{attribute 'GeneratedUsingTerminal: EK1100-0000-0018'}
{attribute addProperty BoxType "EK1100-0000-0018"}
{attribute addProperty Id "RC20_B1_EL7041_1000EL7041_86DE63E743RC20_B2_EL7041_1000EL7041_86DE63E743RC20_C11_EL7041_1000EL7041_86DE63E743RC20_C12_EL7041_1000EL7041_86DE63E743RC20_C21_EL7041_1000EL7041_86DE63E743RC20_C22_EL7041_1000EL7041_86DE63E743RC20_2_EndTerminal_EL9010EL9010_D29C20850"}
{attribute addProperty CRC "1588311305"}
{attribute addProperty Size "258"}
{attribute addProperty Name "RC20_2 (EK1100)"}
TYPE RC20_2_EK1100_5EABB509 EXTENDS EK1100_1FC0878B :
STRUCT
	{attribute addProperty Name "RC20_B1 (EL7041-1000)"}
	{attribute addProperty PreviousPort "RC20_2 (EK1100) : B"}
	RC20_B1_EL7041_1000 : EL7041_86DE63E7;
	{attribute addProperty Name "RC20_B2 (EL7041-1000)"}
	{attribute addProperty PreviousPort "RC20_B1 (EL7041-1000) : B"}
	RC20_B2_EL7041_1000 : EL7041_86DE63E7;
	{attribute addProperty Name "RC20_C11 (EL7041-1000)"}
	{attribute addProperty PreviousPort "RC20_B2 (EL7041-1000) : B"}
	RC20_C11_EL7041_1000 : EL7041_86DE63E7;
	{attribute addProperty Name "RC20_C12 (EL7041-1000)"}
	{attribute addProperty PreviousPort "RC20_C11 (EL7041-1000) : B"}
	RC20_C12_EL7041_1000 : EL7041_86DE63E7;
	{attribute addProperty Name "RC20_C21 (EL7041-1000)"}
	{attribute addProperty PreviousPort "RC20_C12 (EL7041-1000) : B"}
	RC20_C21_EL7041_1000 : EL7041_86DE63E7;
	{attribute addProperty Name "RC20_C22 (EL7041-1000)"}
	{attribute addProperty PreviousPort "RC20_C21 (EL7041-1000) : B"}
	RC20_C22_EL7041_1000 : EL7041_86DE63E7;
	{attribute addProperty Name "RC20_2_EndTerminal (EL9010)"}
	{attribute addProperty PreviousPort "RC20_C22 (EL7041-1000) : B"}
	RC20_2_EndTerminal_EL9010 : EL9010_D29C2085;
END_STRUCT
END_TYPE

(* stored: Version 1.2.0.0, ProductVersion 3.1.4024.11
   DUT RC20_2_EK1100_5EABB509: Id {5f0b0e59-238f-0666-379c-3871ebf6e20e} *)
